TYPE ST_Enabeling :
STRUCT
	bWinchEnable : BOOL := FALSE;
	bCylEnable : BOOL := FALSE; 
	bPosEnable : BOOL := FALSE;
	bVelEnable : BOOL := FALSE;
END_STRUCT
END_TYPE

(* stored: Version 1.1.0.1, ProductVersion 3.1.4024.12
   DUT ST_Enabeling: Id {d9d78ccc-bd5a-4d0d-b03b-559056f1c244} *)
